(* IEC 61131-3 sources: CODESYS-IO-Visualization/CODESYS-IO-Visualization.fbsproj/Pi.device.xml.v3^/Plc Logic.plclogic.xml.v3^/Application.application.xml.v3^/Global Vars, 4 files *)

(* ---- Controller.gvl ---- *)
VAR_GLOBAL
	CPU: CodeSysCPU_UDT := (
		Name := "Example CODESYS PLC",
		Description := "Example OOP with Visualization",
		IPAddress_A := "192.168.160.13",
		IPAddress_B := "192.168.0.1",
		CPUType := "Raspberry Pi",
		SlotCount := 8
	);

	ClockLocal: PLCClock_UDT;
	ClockUTC: PLCClock_UDT;

	SimulationRunning: BOOL;
END_VAR

(* ---- IO.gvl ---- *)
VAR_GLOBAL
	Rack_01: Rack_Opto_RIO_UDT := (SlotCount := 8, InUse := TRUE,
		Modules :=
		[
			(SlotNumber := 0, InUse := TRUE, ModuleType := "UIO", ChannelCount := 10, Channels :=
			[
				(ZeroRaw := 1000.0, SpanRaw := 1839.7, Units := "C", ZeroEu := 0.0, SpanEu := 500.0, ChannelType := IOChannelType.ctAI, SignalName := "Ambient_Temp", LoopNumber := "TI-10001", Description := "Ambient Temperature", InvertValue := FALSE),
				(ZeroRaw := 0.0, SpanRaw := 500.0, Units := "C", ZeroEu := 0.0, SpanEu := 500.0, ChannelType := IOChannelType.ctAI, SignalName := "Pump_Temp", LoopNumber := "TI-10002", Description := "Pump 1 Temperature", InvertValue := FALSE),
				(ZeroRaw := 0.0, SpanRaw := 10.0, Units := "%", ZeroEu := 0.0, SpanEu := 100.0, ChannelType := IOChannelType.ctAI, SignalName := "Pump_Speed", LoopNumber := "AI-10003", Description := "Pump 1 Speed", InvertValue := FALSE),
				(ZeroRaw := 0.0, SpanRaw := 10.0, Units := "gpm", ZeroEu := 0.0, SpanEu := 5000.0, ChannelType := IOChannelType.ctAI, SignalName := "Pump_Flow", LoopNumber := "AI-10004", Description := "Pump 1 Flow", InvertValue := FALSE),
				(ZeroRaw := 4.0, SpanRaw := 16.0, Units := "", ZeroEu := 0.0, SpanEu := 100.0, ChannelType := IOChannelType.ctDI, SignalName := "Pump_Stat", LoopNumber := "YRI-10005", Description := "Pump 1 Running", InvertValue := FALSE),
				(ZeroRaw := 4.0, SpanRaw := 16.0, Units := "", ZeroEu := 0.0, SpanEu := 100.0, ChannelType := IOChannelType.ctDI, SignalName := "Pump_Failed", LoopNumber := "YFI-10005", Description := "Pump 1 Failed", InvertValue := FALSE),
				(ZeroRaw := 4.0, SpanRaw := 16.0, Units := "%", ZeroEu := 0.0, SpanEu := 100.0, ChannelType := IOChannelType.ctAO, SignalName := "Pump_Speed_Out", LoopNumber := "AO-10007", Description := "Pump 1 Speed Out", InvertValue := FALSE),
				(ZeroRaw := 4.0, SpanRaw := 16.0, Units := "gpm", ZeroEu := 0.0, SpanEu := 5000.0, ChannelType := IOChannelType.ctAO, SignalName := "Pump_Flow_Out", LoopNumber := "AO-10008", Description := "Pump 1 Flow Out", InvertValue := FALSE),
				(ZeroRaw := 4.0, SpanRaw := 16.0, Units := "", ZeroEu := 0.0, SpanEu := 100.0, ChannelType := IOChannelType.ctDO, SignalName := "Pump_Running_Out", LoopNumber := "DO-10009", Description := "Pump 1 Running Out", InvertValue := FALSE),
				(ZeroRaw := 4.0, SpanRaw := 16.0, Units := "", ZeroEu := 0.0, SpanEu := 100.0, ChannelType := IOChannelType.ctDO, SignalName := "Pump_Failed_Out", LoopNumber := "DO-10010", Description := "Pump 1 Failed Out", InvertValue := FALSE)
			]),

			(SlotNumber := 1, InUse := FALSE, ModuleType := "NA", ChannelCount := 0),

			(SlotNumber := 2, InUse := FALSE, ModuleType := "NA", ChannelCount := 0),

			(SlotNumber := 3, InUse := FALSE, ModuleType := "NA", ChannelCount := 0),

			(SlotNumber := 4, InUse := FALSE, ModuleType := "NA", ChannelCount := 0),

			(SlotNumber := 5, InUse := FALSE, ModuleType := "NA", ChannelCount := 0),

			(SlotNumber := 6, InUse := FALSE, ModuleType := "NA", ChannelCount := 0),

			(SlotNumber := 7, InUse := FALSE, ModuleType := "NA", ChannelCount := 0)
		]
	);

	Pump_Inlet_Valve_MB: RotorkValve_UDT := (Description := "Pump 1 Inlet Valve", LoopNumber := "CV-01",IPAddress := "192.168.160.39", SimulationEnable := TRUE);
	Pump_Inlet_Valve_In: RotorkValve_MBIO_InputData_UDT;
	Pump_Inlet_Valve_Out: RotorkValve_MBIO_OutputData_UDT;

	Pump_Outlet_Valve_MB: RotorkValve_UDT := (Description := "Pump 1 Outlet Valve", LoopNumber := "CV-02",IPAddress := "192.168.160.39", SimulationEnable := TRUE);
	Pump_Outlet_Valve_In: RotorkValve_MBIO_InputData_UDT;
	Pump_Outlet_Valve_Out: RotorkValve_MBIO_OutputData_UDT;
END_VAR

(* ---- Simulation.gvl ---- *)
{attribute 'qualified_only'}
VAR_GLOBAL
	SimulationEnable: BOOL;
END_VAR

(* ---- Site.gvl ---- *)
VAR_GLOBAL

	Plant: Plant_UDT :=
	(

		AmbientTemp :=
		(
			TagDesc := "Ambient Temperature", TagNo := "TI-10001",
			CurVal := (EU := "C", LowRange :=  0.0, HighRange :=  500.0),
			CurVal2 := (EU := "F", LowRange :=  32.0, HighRange :=  932.0, Offset :=  32.0, Multiplier :=  1.8, Mode := 1, InUse := TRUE),
			DeviceFail := (Enable := TRUE, Description := "Failed", EnableLatch := FALSE, Setpoint := TRUE, OnTimer := (PT :=  1.0), OffTimer := (PT :=  0.0)),
			HiHi := (Enable := TRUE, Description := "HiHi", EnableLatch := FALSE, Rising := TRUE, Setpoint :=  30.0, Deadband :=  1.0, OnTimer := (PT :=  1.0), OffTimer := (PT :=  0.0)),
			Hi := (Enable := TRUE, Description := "Hi", EnableLatch := FALSE, Rising := TRUE, Setpoint :=  28.0, Deadband :=  1.0, OnTimer := (PT :=  1.0), OffTimer := (PT :=  0.0)),
			Lo := (Enable := TRUE, Description := "Lo", EnableLatch := FALSE, Rising := FALSE, Setpoint :=  15.0, Deadband :=  1.0, OnTimer := (PT :=  1.0), OffTimer := (PT :=  0.0)),
			LoLo := (Enable := TRUE, Description := "LoLo", EnableLatch := FALSE, Rising := FALSE, Setpoint :=  13.0, Deadband :=  1.0, OnTimer := (PT :=  1.0), OffTimer := (PT :=  0.0))
		),

		Pump1 :=
		(

			Temp :=
			(
				TagDesc := "Pump 1 Temperature", TagNo := "TI-10002",
				CurVal := (EU := "C", LowRange :=  0.0, HighRange :=  500.0),
				CurVal2 := (EU := "F", LowRange :=  32.0, HighRange :=  932.0, Offset :=  32.0, Multiplier :=  1.8, Mode := 1, InUse := TRUE),
				DeviceFail := (Enable := TRUE, Description := "Failed", EnableLatch := FALSE, Setpoint := TRUE, OnTimer := (PT :=  1.0), OffTimer := (PT :=  0.0)),
				HiHi := (Enable := TRUE, Description := "HiHi", EnableLatch := FALSE, Rising := TRUE, Setpoint :=  150.0, Deadband :=  1.0, OnTimer := (PT :=  1.0), OffTimer := (PT :=  0.0)),
				Hi := (Enable := TRUE, Description := "Hi", EnableLatch := FALSE, Rising := TRUE, Setpoint :=  160.0, Deadband :=  1.0, OnTimer := (PT :=  1.0), OffTimer := (PT :=  0.0)),
				Lo := (Enable := TRUE, Description := "Lo", EnableLatch := FALSE, Rising := FALSE, Setpoint :=  20.0, Deadband :=  1.0, OnTimer := (PT :=  1.0), OffTimer := (PT :=  0.0)),
				LoLo := (Enable := TRUE, Description := "LoLo", EnableLatch := FALSE, Rising := FALSE, Setpoint :=  18.0, Deadband :=  1.0, OnTimer := (PT :=  1.0), OffTimer := (PT :=  0.0))
			),

			Flow :=
			(
				TagDesc := "Pump 1 Flow", TagNo := "AI-10004",
				CurVal := (EU := "gpm", LowRange :=  0.0, HighRange :=  5000.0, ClampLowEnable := TRUE, ClampLow := 10.0),
				CurVal2 := (EU := "mgd", LowRange :=  0.0, HighRange :=  7.2, Offset :=  0.0, Multiplier :=  0.00144, Mode := 1, InUse := TRUE),
				DeviceFail := (Enable := TRUE, Description := "Failed", EnableLatch := FALSE, Setpoint := TRUE, OnTimer := (PT :=  1.0), OffTimer := (PT :=  0.0)),
				DeviceWarning := (Enable := TRUE, Description := "Warning", EnableLatch := FALSE, Setpoint := TRUE, OnTimer := (PT :=  1.0), OffTimer := (PT :=  0.0)),
				HiHi := (Enable := TRUE, Description := "HiHi", Rising := TRUE, Setpoint :=  4500.0, Deadband :=  10.0, OnTimer := (PT :=  1.0), OffTimer := (PT :=  0.0)),
				Hi := (Enable := TRUE, Description := "Hi", Rising := TRUE, Setpoint :=  4000.0, Deadband :=  10.0, OnTimer := (PT :=  1.0), OffTimer := (PT :=  0.0)),
				Accum :=
				[
					(Enable := TRUE, Period := 2, Gain :=  0.000001, Timebase := 60.0, ZeroLimit :=  0.01, EU := "mg", Description := "Daily Total", MaxTotalChange := 10.0, Mode := 0),
					(Enable := TRUE, Period := 3, Gain :=  0.000001, Timebase := 60.0, ZeroLimit :=  0.01, EU := "mg", Description := "Monthly Total", MaxTotalChange := 10.0, Mode := 0),
					(Enable := TRUE, Period := 0, Gain :=  0.000001, Timebase := 60.0, ZeroLimit :=  0.01, EU := "mg", Description := "Total", MaxTotalChange := 10.0, Mode := 0)
				]
			),

			InletValve :=
			(
				TagDesc := "Pump 1 Inlet Valve", TagNo := "CV-01",
				Failure :=
				[
					(Enable := TRUE, Description := "Valve Failed", EnableLatch := TRUE, Setpoint := TRUE, OnTimer := (PT :=  1.0), OffTimer := (PT :=  0.0)),
					(Enable := TRUE, Description := "Valve Overload", EnableLatch := TRUE, Setpoint := TRUE, OnTimer := (PT :=  1.0), OffTimer := (PT :=  0.0)),
					(Enable := TRUE, Description := "Valve Communications Failure", EnableLatch := FALSE, Setpoint := TRUE, OnTimer := (PT :=  1.0), OffTimer := (PT :=  0.0))
				],
				Warning :=
				[
					(Enable := TRUE, Description := "Valve Alarm", EnableLatch := FALSE, Setpoint := TRUE, OnTimer := (PT :=  1.0), OffTimer := (PT :=  0.0))
				],
				Interlock :=
				[
					(Enable := TRUE, Description := "Valve Interlock", EnableLatch := FALSE, Setpoint := TRUE, OnTimer := (PT :=  1.0), OffTimer := (PT :=  0.0))
				],
				NotReady :=
				[
					(Enable := TRUE, Description := "Not in Auto", EnableLatch := FALSE, Setpoint := FALSE, OnTimer := (PT :=  1.0), OffTimer := (PT :=  0.0))
				]
			),

			OutletValve :=
			(
				TagDesc := "Pump 1 Outlet Valve", TagNo := "CV-02",
				Failure :=
				[
					(Enable := TRUE, Description := "Valve Failed", EnableLatch := TRUE, Setpoint := TRUE, OnTimer := (PT :=  1.0), OffTimer := (PT :=  0.0)),
					(Enable := TRUE, Description := "Valve Overload", EnableLatch := TRUE, Setpoint := TRUE, OnTimer := (PT :=  1.0), OffTimer := (PT :=  0.0)),
					(Enable := TRUE, Description := "Valve Communications Failure", EnableLatch := FALSE, Setpoint := TRUE, OnTimer := (PT :=  1.0), OffTimer := (PT :=  0.0))
				],
				Warning :=
				[
					(Enable := TRUE, Description := "Valve Alarm", EnableLatch := FALSE, Setpoint := TRUE, OnTimer := (PT :=  1.0), OffTimer := (PT :=  0.0))
				],
				Interlock :=
				[
					(Enable := TRUE, Description := "Valve Interlock", EnableLatch := FALSE, Setpoint := TRUE, OnTimer := (PT :=  1.0), OffTimer := (PT :=  0.0))
				],
				NotReady :=
				[
					(Enable := TRUE, Description := "Not in Auto", EnableLatch := FALSE, Setpoint := FALSE, OnTimer := (PT :=  1.0), OffTimer := (PT :=  0.0))
				]
			),

			VFD :=
			(
				TagDesc := "Pump 1 VFD", TagNo := "VFD-01",
				PIDSettings1 := (InUse := TRUE, P :=  3.0, I :=  0.5, D :=  0.0, DB :=  1.0, DB_Enable := FALSE, Description := "Flow PID Settings"),
				PID := (irLoLimitSP := 0.0, irHiLimitSP := 5000.0),
				Failure :=
				[
					(Enable := TRUE, Description := "VFD Fault", EnableLatch := FALSE, Setpoint := TRUE, OnTimer := (PT :=  1.0), OffTimer := (PT :=  0.0))
				],
				Timer0 :=
				[
					(PT := 2.0)
				]
			)
		)
	);
END_VAR
